// Type alias for an array iterator.
TYPE T_ArrayIterator : ST_ArrayIterator; END_TYPE

(* stored: Version 1.1.0.1
   DUT T_ArrayIterator: Id {207c955e-dbdb-0288-3eb0-6311a20e5525} *)
